TYPE SideClampVar :
STRUCT
    sv_bButtonFwd: BOOL;
	sv_bButtonBwd: BOOL;
END_STRUCT
END_TYPE

(* stored: Version 1.1.0.1, ProductVersion 3.1.4024.15
   DUT SideClampVar: Id {be9d3f90-baa8-4a51-9c57-29156999b4d9} *)
